// TIA Portal V20 export
DATA_BLOCK "Instance_FB_Get_Out_Rework_Conveyor_Belt_DB"   // DB109
// stored: AutoNumber false, InstanceOfName FB_Get_Out_Rework_Conveyor_Belt, InstanceOfType FB
"FB_Get_Out_Rework_Conveyor_Belt"
   // VAR_INPUT
   //    Emergency_Stop_Release : Bool;
   //    Sensor_Water_Fountain_Geting_Exit_Rework_Conveyor_Belt : Bool;
   //    Button_Water_Fountain_Get_Exit_Rework_Conveyor_Belt : Bool;
   //    Sensor_Spinner_Entrace_Functional_Test_Position_Advanced : Bool;
   //    Sensor_Water_Fountain_Entrace_Functional_Test_Spinner_Conveyor_Belt : Bool;
   // END_VAR
   // VAR_OUTPUT
   //    Turn_On_Conveyor_Belt_Motor_Rework_Conveyor_Belt_Get_Entrace_Functional_Test : Bool;
   // END_VAR
   // VAR
   //    Aux_Trig_0 : Bool;
   //    Aux_Trig_1 : Bool;
   //    Aux_Trig_2 : Bool;
   //    Aux_Trig_3 : Bool;
   //    Aux_Trig_4 : Bool;
   //    Aux_Trig_5 : Bool;
   //    Aux_Trig_6 : Bool;
   //    Aux_Trig_7 : Bool;
   //    Button_Is_Pressed : Bool;
   // END_VAR
BEGIN
END_DATA_BLOCK
